TYPE E_WeekDay :
	(domingo:=0,
	segunda:=1,
	terca:=2,
	quarta:=3,
	quinta:=4,
	sexta:=5,
	sabado:=6);
END_TYPE

(* stored: Version 1.1.0.1, ProductVersion 3.1.4020.6
   DUT E_WeekDay: Id {8818f059-54ea-4eb9-a561-ab55ecb88770} *)
